// TwinCAT 3 PLC project main
// ProgramVersion: 3.1.4024.0
// libraries:
//   Tc2_Standard, * (Beckhoff Automation GmbH)
//   Tc2_System, * (Beckhoff Automation GmbH)
//   Tc3_Module, * (Beckhoff Automation GmbH)
// project tree:
//   / GlobalTextList.TcGTLO, PlcTask.TcTTO, Visualization Manager.TcVMO (not stored)
//   POUs/ MAIN.TcPOU
//   VISUs/ Visu.TcVIS
// real-time tasks:
//   TASK PlcTask: cycle T#10ms, priority 20, ADS port 350

CONFIGURATION main
    RESOURCE PLC ON TwinCAT3
        TASK PlcTask(INTERVAL := T#10ms, PRIORITY := 20);
        PROGRAM MAIN WITH PlcTask : MAIN;
    END_RESOURCE
END_CONFIGURATION

// ---- POUs/MAIN.TcPOU
PROGRAM MAIN
VAR
	bS01 : BOOL;
	bS02 : BOOL;
	bS03 : BOOL;
	bS04 : BOOL;
	bS05 : BOOL;
	
	bQ01 : BOOL;
	bQ02 : BOOL;
	bQ03 : bool;
END_VAR

bQ01 := bS01 AND ((bS03 OR bS04 OR bS05) OR (bS03 AND bS04 AND bS05));
bQ02 := bS01 AND ((bS03 AND bS04) OR (bS03 AND bS05) OR (bS04 AND bS05) OR (bS03 AND bS04 AND bS05));
bQ03 := bS01 AND (bS03 AND bS04 AND bS05) AND NOT bS02;

END_PROGRAM

// ---- GlobalTextList.TcGTLO
TEXTLIST GlobalTextList
  537 = 'bQ01'
  256 = 'bQ02'
  9 = 'bQ03'
  576 = 'bS01'
  896 = 'bS02'
  573 = 'bS03'
  849 = 'bS04'
  999 = 'bS05'
END_TEXTLIST

// ---- VISUs/Visu.TcVIS
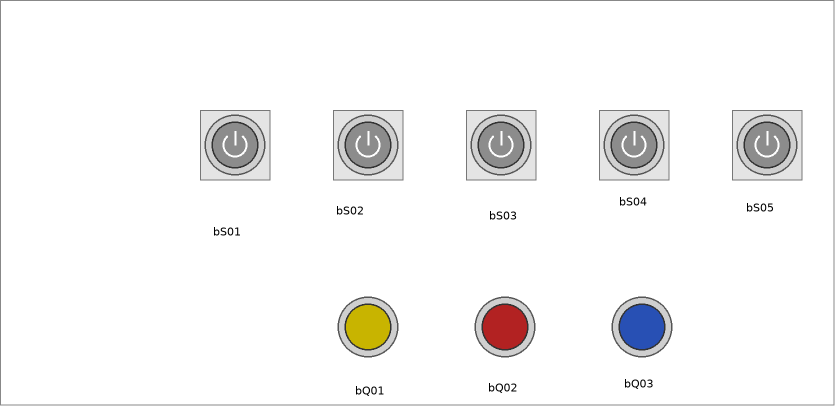
VISUALIZATION Visu  // 835x406
    PowerSwitch (200,110 70x70), variable: MAIN.bS01, behaviour: TOGGLE, style: Switch-PowerSwitch-Gray
    PowerSwitch (333,110 70x70), variable: MAIN.bS02, behaviour: TOGGLE, style: Switch-PowerSwitch-Gray
    PowerSwitch (466,110 70x70), variable: MAIN.bS03, behaviour: TOGGLE, style: Switch-PowerSwitch-Gray
    PowerSwitch (599,110 70x70), variable: MAIN.bS04, behaviour: TOGGLE, style: Switch-PowerSwitch-Gray
    PowerSwitch (732,110 70x70), variable: MAIN.bS05, behaviour: TOGGLE, style: Switch-PowerSwitch-Gray
    Lamp1 (333,292 70x70), variable: MAIN.bQ01, style: Lamp-Lamp1-Yellow
    Lamp1 (470,292 70x70), variable: MAIN.bQ02, style: Lamp-Lamp1-Red
    Lamp1 (607,292 70x70), variable: MAIN.bQ03, style: Lamp-Lamp1-Blue
    Label (152,217 150x30), "bS01"
    Label (275,196 150x30), "bS02"
    Label (564,369 150x30), "bQ03"
    Label (428,373 150x30), "bQ02"
    Label (295,376 150x30), "bQ01"
    Label (428,201 150x30), "bS03"
    Label (558,187 150x30), "bS04"
    Label (685,193 150x30), "bS05"
END_VISUALIZATION
